{attribute 'qualified_only'}
{attribute 'strict'}
TYPE E_State_Can_Supply :
(
	State := 0
);
END_TYPE

(* stored: Version 1.1.0.1, ProductVersion 3.1.4024.12
   DUT E_State_Can_Supply: Id {af5490b1-04dd-43b4-b9e7-2ad3b212618a} *)
